// TwinCAT 3 PLC project Untitled1
// ProgramVersion: 3.1.4024.0
// libraries:
//   Tc2_Standard, * (Beckhoff Automation GmbH)
//   Tc2_System, * (Beckhoff Automation GmbH)
//   Tc3_Module, * (Beckhoff Automation GmbH)
//   Tc3_Vision, * (Beckhoff Automation GmbH)
// project tree:
//   / PlcTask.TcTTO
//   POUs/ MAIN.TcPOU

CONFIGURATION Untitled1
    RESOURCE PLC ON TwinCAT3
        TASK PlcTask(INTERVAL := T#10ms, PRIORITY := 20);
        PROGRAM MAIN WITH PlcTask : MAIN;
    END_RESOURCE
END_CONFIGURATION

// ---- POUs/MAIN.TcPOU
PROGRAM MAIN
VAR
    CycleCount       : UDINT;
    hr               : HRESULT;
    fbCamera         : FB_VN_FileSourceControl;
    eState           : ETcVnCameraState;
    ipImageIn        : ITcVnImage;
    ipImageInDisp    : ITcVnDisplayableImage;
    nNewImageCounter : UINT;
    sText            : STRING;
    aColorBlack      : TcVnVector4_LREAL := [0, 0, 0, 255];
END_VAR

CycleCount := CycleCount + 1;

eState := fbCamera.GetState();

IF eState = TCVN_CS_ERROR THEN
    hr := fbCamera.Reset();

ELSIF eState < TCVN_CS_ACQUIRING THEN
    hr := fbCamera.StartAcquisition();

ELSIF eState = TCVN_CS_ACQUIRING THEN
    hr := fbCamera.GetCurrentImage(ipImageIn);

    // Check if new Image was received
    IF SUCCEEDED(hr) AND ipImageIn <> 0 THEN
        nNewImageCounter := nNewImageCounter + 1;
        sText            := UDINT_TO_STRING(CycleCount);
        hr               := F_VN_PutText(sText,
                                         ipImageIn,
                                         12,
                                         100,
                                         ETcVnFontType.TCVN_FT_HERSHEY_PLAIN,
                                         2,
                                         aColorBlack,
                                         hr);

        // Place to call vision algorithms
        hr := F_VN_TransformIntoDisplayableImage(ipImageIn, ipImageInDisp, hr);
    END_IF
END_IF

END_PROGRAM
